FUNCTION_BLOCK EspPayloadDecoder IMPLEMENTS ITF_PayloadDecoder
VAR
END_VAR

END_FUNCTION_BLOCK

(* stored: Version 1.1.0.1
   POU EspPayloadDecoder: Id {3c23ce38-a44c-4571-993b-09ac9f9fd58b}, SpecialFunc None *)
